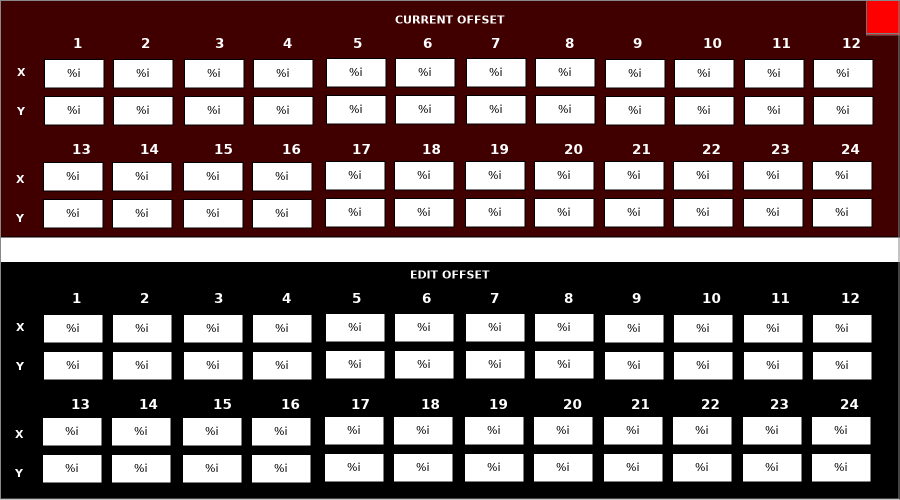
VISUALIZATION MOffset_3  // 900x500
    RoundedRectangle (0,0 900x237)
    Label (0,0 900x40), "CURRENT OFFSET"
    Label (14,55 25x35), "X"
    RoundedRectangle (44,59 60x29), "%i", text variable: Status_GVL.RecipeLine[3].OffsetPattern.Offset_X[1]
    Label (70,26 25x35), "1"
    RoundedRectangle (113,59 60x29), "%i", text variable: Status_GVL.RecipeLine[3].OffsetPattern.Offset_X[2]
    Label (138,26 25x35), "2"
    RoundedRectangle (184,59 60x29), "%i", text variable: Status_GVL.RecipeLine[3].OffsetPattern.Offset_X[3]
    RoundedRectangle (253,59 60x29), "%i", text variable: Status_GVL.RecipeLine[3].OffsetPattern.Offset_X[4]
    Label (14,94 25x35), "Y"
    RoundedRectangle (326,58 60x29), "%i", text variable: Status_GVL.RecipeLine[3].OffsetPattern.Offset_X[5]
    RoundedRectangle (395,58 60x29), "%i", text variable: Status_GVL.RecipeLine[3].OffsetPattern.Offset_X[6]
    RoundedRectangle (466,58 60x29), "%i", text variable: Status_GVL.RecipeLine[3].OffsetPattern.Offset_X[7]
    RoundedRectangle (535,58 60x29), "%i", text variable: Status_GVL.RecipeLine[3].OffsetPattern.Offset_X[8]
    RoundedRectangle (605,59 60x29), "%i", text variable: Status_GVL.RecipeLine[3].OffsetPattern.Offset_X[9]
    RoundedRectangle (674,59 60x29), "%i", text variable: Status_GVL.RecipeLine[3].OffsetPattern.Offset_X[10]
    Label (212,26 25x35), "3"
    Label (280,26 25x35), "4"
    Label (350,26 25x35), "5"
    Label (420,26 25x35), "6"
    Label (488,26 25x35), "7"
    Label (562,26 25x35), "8"
    Label (630,26 25x35), "9"
    Label (700,26 25x35), "10"
    RoundedRectangle (44,96 60x29), "%i", text variable: Status_GVL.RecipeLine[3].OffsetPattern.Offset_Y[1]
    RoundedRectangle (113,96 60x29), "%i", text variable: Status_GVL.RecipeLine[3].OffsetPattern.Offset_Y[2]
    RoundedRectangle (184,96 60x29), "%i", text variable: Status_GVL.RecipeLine[3].OffsetPattern.Offset_Y[3]
    RoundedRectangle (253,96 60x29), "%i", text variable: Status_GVL.RecipeLine[3].OffsetPattern.Offset_Y[4]
    RoundedRectangle (326,95 60x29), "%i", text variable: Status_GVL.RecipeLine[3].OffsetPattern.Offset_Y[5]
    RoundedRectangle (395,95 60x29), "%i", text variable: Status_GVL.RecipeLine[3].OffsetPattern.Offset_Y[6]
    RoundedRectangle (466,95 60x29), "%i", text variable: Status_GVL.RecipeLine[3].OffsetPattern.Offset_Y[7]
    RoundedRectangle (535,95 60x29), "%i", text variable: Status_GVL.RecipeLine[3].OffsetPattern.Offset_Y[8]
    RoundedRectangle (605,96 60x29), "%i", text variable: Status_GVL.RecipeLine[3].OffsetPattern.Offset_Y[9]
    RoundedRectangle (674,96 60x29), "%i", text variable: Status_GVL.RecipeLine[3].OffsetPattern.Offset_Y[10]
    Label (13,162 25x35), "X"
    RoundedRectangle (43,162 60x29), "%i", text variable: Status_GVL.RecipeLine[3].OffsetPattern.Offset_X[13]
    RoundedRectangle (112,162 60x29), "%i", text variable: Status_GVL.RecipeLine[3].OffsetPattern.Offset_X[14]
    RoundedRectangle (183,162 60x29), "%i", text variable: Status_GVL.RecipeLine[3].OffsetPattern.Offset_X[15]
    RoundedRectangle (252,162 60x29), "%i", text variable: Status_GVL.RecipeLine[3].OffsetPattern.Offset_X[16]
    Label (13,201 25x35), "Y"
    RoundedRectangle (325,161 60x29), "%i", text variable: Status_GVL.RecipeLine[3].OffsetPattern.Offset_X[17]
    RoundedRectangle (394,161 60x29), "%i", text variable: Status_GVL.RecipeLine[3].OffsetPattern.Offset_X[18]
    RoundedRectangle (465,161 60x29), "%i", text variable: Status_GVL.RecipeLine[3].OffsetPattern.Offset_X[19]
    RoundedRectangle (534,161 60x29), "%i", text variable: Status_GVL.RecipeLine[3].OffsetPattern.Offset_X[20]
    RoundedRectangle (604,161 60x29), "%i", text variable: Status_GVL.RecipeLine[3].OffsetPattern.Offset_X[21]
    RoundedRectangle (673,161 60x29), "%i", text variable: Status_GVL.RecipeLine[3].OffsetPattern.Offset_X[22]
    RoundedRectangle (43,199 60x29), "%i", text variable: Status_GVL.RecipeLine[3].OffsetPattern.Offset_Y[13]
    RoundedRectangle (112,199 60x29), "%i", text variable: Status_GVL.RecipeLine[3].OffsetPattern.Offset_Y[14]
    RoundedRectangle (183,199 60x29), "%i", text variable: Status_GVL.RecipeLine[3].OffsetPattern.Offset_Y[15]
    RoundedRectangle (252,199 60x29), "%i", text variable: Status_GVL.RecipeLine[3].OffsetPattern.Offset_Y[16]
    RoundedRectangle (325,198 60x29), "%i", text variable: Status_GVL.RecipeLine[3].OffsetPattern.Offset_Y[17]
    RoundedRectangle (394,198 60x29), "%i", text variable: Status_GVL.RecipeLine[3].OffsetPattern.Offset_Y[18]
    RoundedRectangle (465,198 60x29), "%i", text variable: Status_GVL.RecipeLine[3].OffsetPattern.Offset_Y[19]
    RoundedRectangle (534,198 60x29), "%i", text variable: Status_GVL.RecipeLine[3].OffsetPattern.Offset_Y[20]
    RoundedRectangle (604,198 60x29), "%i", text variable: Status_GVL.RecipeLine[3].OffsetPattern.Offset_Y[21]
    RoundedRectangle (673,198 60x29), "%i", text variable: Status_GVL.RecipeLine[3].OffsetPattern.Offset_Y[22]
    Label (69,132 25x35), "13"
    Label (137,132 25x35), "14"
    Label (211,132 25x35), "15"
    Label (279,132 25x35), "16"
    Label (349,132 25x35), "17"
    Label (419,132 25x35), "18"
    Label (487,132 25x35), "19"
    Label (561,132 25x35), "20"
    Label (629,132 25x35), "21"
    Label (699,132 25x35), "22"
    RoundedRectangle (0,262 900x237)
    Label (0,255 900x40), "EDIT OFFSET"
    Label (13,310 25x35), "X"
    RoundedRectangle (43,314 60x29), "%i", text variable: HMI_GVL.arRecipeHMI[3].OffsetPattern.Offset_X[1], input disabled if: Status_GVL.StsEdit[3]
        OnMouseClick: write the text variable via Default
    Label (69,281 25x35), "1"
    RoundedRectangle (112,314 60x29), "%i", text variable: HMI_GVL.arRecipeHMI[3].OffsetPattern.Offset_X[2], input disabled if: Status_GVL.StsEdit[3]
        OnMouseClick: write the text variable via Default
    Label (137,281 25x35), "2"
    RoundedRectangle (183,314 60x29), "%i", text variable: HMI_GVL.arRecipeHMI[3].OffsetPattern.Offset_X[3], input disabled if: Status_GVL.StsEdit[3]
        OnMouseClick: write the text variable via Default
    RoundedRectangle (252,314 60x29), "%i", text variable: HMI_GVL.arRecipeHMI[3].OffsetPattern.Offset_X[4], input disabled if: Status_GVL.StsEdit[3]
        OnMouseClick: write the text variable via Default
    Label (13,349 25x35), "Y"
    RoundedRectangle (325,313 60x29), "%i", text variable: HMI_GVL.arRecipeHMI[3].OffsetPattern.Offset_X[5], input disabled if: Status_GVL.StsEdit[3]
        OnMouseClick: write the text variable via Default
    RoundedRectangle (394,313 60x29), "%i", text variable: HMI_GVL.arRecipeHMI[3].OffsetPattern.Offset_X[6], input disabled if: Status_GVL.StsEdit[3]
        OnMouseClick: write the text variable via Default
    RoundedRectangle (465,313 60x29), "%i", text variable: HMI_GVL.arRecipeHMI[3].OffsetPattern.Offset_X[7], input disabled if: Status_GVL.StsEdit[3]
        OnMouseClick: write the text variable via Default
    RoundedRectangle (534,313 60x29), "%i", text variable: HMI_GVL.arRecipeHMI[3].OffsetPattern.Offset_X[8], input disabled if: Status_GVL.StsEdit[3]
        OnMouseClick: write the text variable via Default
    RoundedRectangle (604,314 60x29), "%i", text variable: HMI_GVL.arRecipeHMI[3].OffsetPattern.Offset_X[9], input disabled if: Status_GVL.StsEdit[3]
        OnMouseClick: write the text variable via Default
    RoundedRectangle (673,314 60x29), "%i", text variable: HMI_GVL.arRecipeHMI[3].OffsetPattern.Offset_X[10], input disabled if: Status_GVL.StsEdit[3]
        OnMouseClick: write the text variable via Default
    Label (211,281 25x35), "3"
    Label (279,281 25x35), "4"
    Label (349,281 25x35), "5"
    Label (419,281 25x35), "6"
    Label (487,281 25x35), "7"
    Label (561,281 25x35), "8"
    Label (629,281 25x35), "9"
    Label (699,281 25x35), "10"
    RoundedRectangle (43,351 60x29), "%i", text variable: HMI_GVL.arRecipeHMI[3].OffsetPattern.Offset_Y[1], input disabled if: Status_GVL.StsEdit[3]
        OnMouseClick: write the text variable via Default
    RoundedRectangle (112,351 60x29), "%i", text variable: HMI_GVL.arRecipeHMI[3].OffsetPattern.Offset_Y[2], input disabled if: Status_GVL.StsEdit[3]
        OnMouseClick: write the text variable via Default
    RoundedRectangle (183,351 60x29), "%i", text variable: HMI_GVL.arRecipeHMI[3].OffsetPattern.Offset_Y[3], input disabled if: Status_GVL.StsEdit[3]
        OnMouseClick: write the text variable via Default
    RoundedRectangle (252,351 60x29), "%i", text variable: HMI_GVL.arRecipeHMI[3].OffsetPattern.Offset_Y[4], input disabled if: Status_GVL.StsEdit[3]
        OnMouseClick: write the text variable via Default
    RoundedRectangle (325,350 60x29), "%i", text variable: HMI_GVL.arRecipeHMI[3].OffsetPattern.Offset_Y[5], input disabled if: Status_GVL.StsEdit[3]
        OnMouseClick: write the text variable via Default
    RoundedRectangle (394,350 60x29), "%i", text variable: HMI_GVL.arRecipeHMI[3].OffsetPattern.Offset_Y[6], input disabled if: Status_GVL.StsEdit[3]
        OnMouseClick: write the text variable via Default
    RoundedRectangle (465,350 60x29), "%i", text variable: HMI_GVL.arRecipeHMI[3].OffsetPattern.Offset_Y[7], input disabled if: Status_GVL.StsEdit[3]
        OnMouseClick: write the text variable via Default
    RoundedRectangle (534,350 60x29), "%i", text variable: HMI_GVL.arRecipeHMI[3].OffsetPattern.Offset_Y[8], input disabled if: Status_GVL.StsEdit[3]
        OnMouseClick: write the text variable via Default
    RoundedRectangle (604,351 60x29), "%i", text variable: HMI_GVL.arRecipeHMI[3].OffsetPattern.Offset_Y[9], input disabled if: Status_GVL.StsEdit[3]
        OnMouseClick: write the text variable via Default
    RoundedRectangle (673,351 60x29), "%i", text variable: HMI_GVL.arRecipeHMI[3].OffsetPattern.Offset_Y[10], input disabled if: Status_GVL.StsEdit[3]
        OnMouseClick: write the text variable via Default
    Label (12,417 25x35), "X"
    RoundedRectangle (42,417 60x29), "%i", text variable: HMI_GVL.arRecipeHMI[3].OffsetPattern.Offset_X[13], input disabled if: Status_GVL.StsEdit[3]
        OnMouseClick: write the text variable via Default
    RoundedRectangle (111,417 60x29), "%i", text variable: HMI_GVL.arRecipeHMI[3].OffsetPattern.Offset_X[14], input disabled if: Status_GVL.StsEdit[3]
        OnMouseClick: write the text variable via Default
    RoundedRectangle (182,417 60x29), "%i", text variable: HMI_GVL.arRecipeHMI[3].OffsetPattern.Offset_X[15], input disabled if: Status_GVL.StsEdit[3]
        OnMouseClick: write the text variable via Default
    RoundedRectangle (251,417 60x29), "%i", text variable: HMI_GVL.arRecipeHMI[3].OffsetPattern.Offset_X[16], input disabled if: Status_GVL.StsEdit[3]
        OnMouseClick: write the text variable via Default
    Label (12,456 25x35), "Y"
    RoundedRectangle (324,416 60x29), "%i", text variable: HMI_GVL.arRecipeHMI[3].OffsetPattern.Offset_X[17], input disabled if: Status_GVL.StsEdit[3]
        OnMouseClick: write the text variable via Default
    RoundedRectangle (393,416 60x29), "%i", text variable: HMI_GVL.arRecipeHMI[3].OffsetPattern.Offset_X[18], input disabled if: Status_GVL.StsEdit[3]
        OnMouseClick: write the text variable via Default
    RoundedRectangle (464,416 60x29), "%i", text variable: HMI_GVL.arRecipeHMI[3].OffsetPattern.Offset_X[19], input disabled if: Status_GVL.StsEdit[3]
        OnMouseClick: write the text variable via Default
    RoundedRectangle (533,416 60x29), "%i", text variable: HMI_GVL.arRecipeHMI[3].OffsetPattern.Offset_X[20], input disabled if: Status_GVL.StsEdit[3]
        OnMouseClick: write the text variable via Default
    RoundedRectangle (603,416 60x29), "%i", text variable: HMI_GVL.arRecipeHMI[3].OffsetPattern.Offset_X[21], input disabled if: Status_GVL.StsEdit[3]
        OnMouseClick: write the text variable via Default
    RoundedRectangle (672,416 60x29), "%i", text variable: HMI_GVL.arRecipeHMI[3].OffsetPattern.Offset_X[22], input disabled if: Status_GVL.StsEdit[3]
        OnMouseClick: write the text variable via Default
    RoundedRectangle (42,454 60x29), "%i", text variable: HMI_GVL.arRecipeHMI[3].OffsetPattern.Offset_Y[13], input disabled if: Status_GVL.StsEdit[3]
        OnMouseClick: write the text variable via Default
    RoundedRectangle (111,454 60x29), "%i", text variable: HMI_GVL.arRecipeHMI[3].OffsetPattern.Offset_Y[14], input disabled if: Status_GVL.StsEdit[3]
        OnMouseClick: write the text variable via Default
    RoundedRectangle (182,454 60x29), "%i", text variable: HMI_GVL.arRecipeHMI[3].OffsetPattern.Offset_Y[15], input disabled if: Status_GVL.StsEdit[3]
        OnMouseClick: write the text variable via Default
    RoundedRectangle (251,454 60x29), "%i", text variable: HMI_GVL.arRecipeHMI[3].OffsetPattern.Offset_Y[16], input disabled if: Status_GVL.StsEdit[3]
        OnMouseClick: write the text variable via Default
    RoundedRectangle (324,453 60x29), "%i", text variable: HMI_GVL.arRecipeHMI[3].OffsetPattern.Offset_Y[17], input disabled if: Status_GVL.StsEdit[3]
        OnMouseClick: write the text variable via Default
    RoundedRectangle (393,453 60x29), "%i", text variable: HMI_GVL.arRecipeHMI[3].OffsetPattern.Offset_Y[18], input disabled if: Status_GVL.StsEdit[3]
        OnMouseClick: write the text variable via Default
    RoundedRectangle (464,453 60x29), "%i", text variable: HMI_GVL.arRecipeHMI[3].OffsetPattern.Offset_Y[19], input disabled if: Status_GVL.StsEdit[3]
        OnMouseClick: write the text variable via Default
    RoundedRectangle (533,453 60x29), "%i", text variable: HMI_GVL.arRecipeHMI[3].OffsetPattern.Offset_Y[20], input disabled if: Status_GVL.StsEdit[3]
        OnMouseClick: write the text variable via Default
    RoundedRectangle (603,453 60x29), "%i", text variable: HMI_GVL.arRecipeHMI[3].OffsetPattern.Offset_Y[21], input disabled if: Status_GVL.StsEdit[3]
        OnMouseClick: write the text variable via Default
    RoundedRectangle (672,453 60x29), "%i", text variable: HMI_GVL.arRecipeHMI[3].OffsetPattern.Offset_Y[22], input disabled if: Status_GVL.StsEdit[3]
        OnMouseClick: write the text variable via Default
    Label (68,387 25x35), "13"
    Label (136,387 25x35), "14"
    Label (210,387 25x35), "15"
    Label (278,387 25x35), "16"
    Label (348,387 25x35), "17"
    Label (418,387 25x35), "18"
    Label (486,387 25x35), "19"
    Label (560,387 25x35), "20"
    Label (628,387 25x35), "21"
    Label (698,387 25x35), "22"
    Button (866,0 35x35), image: VisuSymbols.Symbols.Wrong
        OnMouseClick: CloseDialog Dialog=MOffset_3, Result=OK, NumpadKeypadSet=True
    RoundedRectangle (744,59 60x29), "%i", text variable: Status_GVL.RecipeLine[3].OffsetPattern.Offset_X[11]
    RoundedRectangle (813,59 60x29), "%i", text variable: Status_GVL.RecipeLine[3].OffsetPattern.Offset_X[12]
    Label (769,26 25x35), "11"
    Label (839,26 25x35), "12"
    RoundedRectangle (744,96 60x29), "%i", text variable: Status_GVL.RecipeLine[3].OffsetPattern.Offset_Y[11]
    RoundedRectangle (813,96 60x29), "%i", text variable: Status_GVL.RecipeLine[3].OffsetPattern.Offset_Y[12]
    RoundedRectangle (743,161 60x29), "%i", text variable: Status_GVL.RecipeLine[3].OffsetPattern.Offset_X[23]
    RoundedRectangle (812,161 60x29), "%i", text variable: Status_GVL.RecipeLine[3].OffsetPattern.Offset_X[24]
    RoundedRectangle (743,198 60x29), "%i", text variable: Status_GVL.RecipeLine[3].OffsetPattern.Offset_Y[23]
    RoundedRectangle (812,198 60x29), "%i", text variable: Status_GVL.RecipeLine[3].OffsetPattern.Offset_Y[24]
    Label (768,132 25x35), "23"
    Label (838,132 25x35), "24"
    RoundedRectangle (743,314 60x29), "%i", text variable: HMI_GVL.arRecipeHMI[3].OffsetPattern.Offset_X[11], input disabled if: Status_GVL.StsEdit[3]
        OnMouseClick: write the text variable via Default
    RoundedRectangle (812,314 60x29), "%i", text variable: HMI_GVL.arRecipeHMI[3].OffsetPattern.Offset_X[12], input disabled if: Status_GVL.StsEdit[3]
        OnMouseClick: write the text variable via Default
    Label (768,281 25x35), "11"
    Label (838,281 25x35), "12"
    RoundedRectangle (743,351 60x29), "%i", text variable: HMI_GVL.arRecipeHMI[3].OffsetPattern.Offset_Y[11], input disabled if: Status_GVL.StsEdit[3]
        OnMouseClick: write the text variable via Default
    RoundedRectangle (812,351 60x29), "%i", text variable: HMI_GVL.arRecipeHMI[3].OffsetPattern.Offset_Y[12], input disabled if: Status_GVL.StsEdit[3]
        OnMouseClick: write the text variable via Default
    RoundedRectangle (742,416 60x29), "%i", text variable: HMI_GVL.arRecipeHMI[3].OffsetPattern.Offset_X[23], input disabled if: Status_GVL.StsEdit[3]
        OnMouseClick: write the text variable via Default
    RoundedRectangle (811,416 60x29), "%i", text variable: HMI_GVL.arRecipeHMI[3].OffsetPattern.Offset_X[24], input disabled if: Status_GVL.StsEdit[3]
        OnMouseClick: write the text variable via Default
    RoundedRectangle (742,453 60x29), "%i", text variable: HMI_GVL.arRecipeHMI[3].OffsetPattern.Offset_Y[23], input disabled if: Status_GVL.StsEdit[3]
        OnMouseClick: write the text variable via Default
    RoundedRectangle (811,453 60x29), "%i", text variable: HMI_GVL.arRecipeHMI[3].OffsetPattern.Offset_Y[24], input disabled if: Status_GVL.StsEdit[3]
        OnMouseClick: write the text variable via Default
    Label (767,387 25x35), "23"
    Label (837,387 25x35), "24"
END_VISUALIZATION

(* stored: Version 1.1.0.1, ProductVersion 3.1.4024.12
   Visu MOffset_3: Id {2300bcd8-c7fb-4cd1-b1f0-53da65d24b2a} *)
